PROGRAM Step_7_Saw_Positioning
VAR
	 i : INT;
	NextTargetLength: INT :=0;
	ActiveLength: INT;
	
	
	ftCutDone: F_TRIG;
	ftGradingEndLimit: F_TRIG;
	rtSawFeedChainHomingSensor : R_TRIG;
	rtGoToPosition : R_TRIG;
	rtExecuteAbs1 : R_TRIG;
	
	
	

	
	LocalSafety_7: BOOL;
END_VAR

//------------------Defaults--------------------

SawFeedChainVFD3FWD := FALSE;


// ---------- Safety ----------

LocalSafety_7 := NOT VFD3Faulted AND SawBlade1MMP AND SawBlade2MMP AND DustCollectorMMP;



IF NOT Permissive OR NOT LocalSafety_7 OR CycleStopPB THEN
    Step7_State := 0;
END_IF

//------------------Triggers------------------------------
ftCutDone(CLK := SawPhotoeye); 
rtGoToPosition(CLK := HMI_GoToPosition);
rtExecuteAbs1(CLK := xExecuteDistanceAbs1);


lrActualPosition := GVL_Axes.Axis1.NcToPlc.ActPos;



IF ftCutDone.Q THEN
    FOR i := 1 TO 4 DO
        FootFIFO[i] := FootFIFO[i + 1];
    END_FOR;
    FootFIFO[5] := 0;
END_IF;




//----------------------------------------Board Transfer---------------------------------


// ---------- Trigger to enter POSITIONING (state 0) ----------
IF ftCutDone.Q OR rtGoToPosition.Q THEN // falling edge on SawPhotoeye or HMI button "go to position" 
    Step7_State := 5;
END_IF






// ---------- State machine ----------
CASE Step7_State OF
	
0: // standby


SawFeedChainVFD3FWD := FALSE;
SawBladesFWD := FALSE;
DustCollectorFWD := FALSE;


IF CycleStartPB THEN
	Step7_State := 5;
END_IF





5:  // POSITIONING DECISION

SawBladesFWD := TRUE;
DustCollectorFWD := TRUE;

lrTargetPosition := FootFIFO[1]; // target position from queue

// If there’s no target length, do nothing
IF FootFIFO[1] = 0 THEN
    SawFeedChainVFD3FWD := FALSE;	
ELSE                  
	// Otherwise, continue with positioning logic
	// call FB every scan (Execute FALSE by default here)
        fbMove_Absolute1(
            Axis         := GVL_Axes.Axis1,
            Execute      := FALSE,
            Position     := lrTargetPosition,
            Velocity     := 3500.0,
            Acceleration := ,
            Deceleration := ,
            Jerk         := ,
            BufferMode   := MC_BufferMode.MC_Aborting,
            Options      := ,
	);

	// 1) Check if already at position
	IF ABS(lrActualPosition - lrTargetPosition) <= PositionTolerance (*LREAL := 0.05; // acceptable error window*) THEN
	// already in position, skip move
     Step7_State := 10; // back to feeding
	ELSE
	// 2) Execute a move if not yet in position
    Step7_State := 15; // Execute absolute trget position
	END_IF;
								
END_IF

10: //busy //running// FEEDING 


xExecuteDistanceAbs1:= FALSE;  


// still call FB to keep status fresh
        fbMove_Absolute1(
            Axis         := GVL_Axes.Axis1,
            Execute      := FALSE,
            Position     := lrTargetPosition,
            Velocity     := 3500.0,
            Acceleration := ,
            Deceleration := ,
            Jerk         := ,
            BufferMode   := MC_BufferMode.MC_Aborting,
            Options      := ,
);


SawFeedChainVFD3FWD := TRUE;
 
  // The edges at top will kick us back to state 0
  // when SawPhotoeye falls or HMI_GoToPos is pressed.
 

 
 15: //ISSUE MOVE (one-scan pulse), then wait for done

 
SawFeedChainVFD3FWD := FALSE;     
xExecuteDistanceAbs1:= TRUE;   // pulse Execute
           
       

// Call the motion block
fbMove_Absolute1(
	Axis         := GVL_Axes.Axis1,
	Execute      := rtExecuteAbs1.Q,
	Position     := lrTargetPosition,
	Velocity     := 3500.0,
	Acceleration := ,
	Deceleration := ,
	Jerk         := ,
	BufferMode   := MC_BufferMode.MC_Aborting,
	Options      := ,
);

// When the move is finished...
IF xMoveAbsDone1 THEN
   Step7_State  := 10;  
END_IF;


       

END_CASE

END_PROGRAM

(* stored: Version 1.1.0.1
   POU Step_7_Saw_Positioning: Id {a65fa5f1-e818-47b1-ba2f-444b9555b8e9}, SpecialFunc None *)
